FUNCTION MapClamp : REAL
VAR_INPUT
	flArg				: LREAL; //fFnGenChanVal
	flInMin				: LREAL;
	flInMax				: LREAL;
	flOutMin			: LREAL;
	flOutMax			: LREAL;
	usiBitDepth			: USINT;
END_VAR
VAR
	flValueRange		: LREAL;
	flOutputIncrement	: LREAL;
	diOutputIncrement	: DINT;
	flUnroundedVal		: LREAL;
	diUnroundedVal		: DINT;
	flMapClampFloor		: LREAL;
	flMapClampTemp		: LREAL;
END_VAR

IF (flInMax - flInMin) <> 0 THEN
	flUnroundedVal := (((flArg - flInMin) * (flOutMax - flOutMin)) / (flInMax - flInMin)) + flOutMin;
END_IF

//Basically a sub-function (possibly could be written as a separate function that is called) to compute the nearest value for the output, based on the user input params
flValueRange	:= flOutMax - flOutMin; //Entire possible range of output values;

flOutputIncrement	:= flValueRange/EXPT(2,usiBitDepth);
diOutputIncrement	:= LREAL_TO_DINT(flOutputIncrement);

diUnroundedVal		:= LREAL_TO_INT(flUnroundedVal);

IF flOutputIncrement <> 0 THEN //avoid div by 0
	flMapClampFloor	:= FLOOR(flUnroundedVal / flOutputIncrement);//Truncate? UnroundedValue, add one increment
END_IF

IF flOutputIncrement <> 0 THEN //avoid div by 0
	IF (diUnroundedVal MOD diOutputIncrement) >= (0.5 * flOutputIncrement) THEN
		MapClamp	:=	(flMapClampFloor * flOutputIncrement) + flOutputIncrement;		//Truncate? UnroundedValue, add one increment 
	ELSIF (diUnroundedVal MOD diOutputIncrement) < (0.5 * flOutputIncrement) THEN
		MapClamp	:=	(flMapClampFloor * flOutputIncrement);
	END_IF
END_IF

IF MapClamp > flOutMax THEN
	MapClamp	:= flOutMax;
ELSIF MapClamp < flOutMin THEN
	MapClamp	:= flOutMin;	
END_IF

END_FUNCTION

(* stored: Version 1.1.0.1, ProductVersion 3.1.4024.6
   POU MapClamp: Id {99180469-7fa6-47c0-b540-696eba09b4bf}, SpecialFunc None *)
